(* CODESYS project Untitled2.project
   CustomField04_name: CustomField04
   CustomField06_name: CustomField06
   CustomField07_name: CustomField07
   CustomField09_name: CustomField09
   CustomField08_name: CustomField08
   CustomField02_name: CustomField02
   CustomField10_name: CustomField10
   CustomField01_name: CustomField01
   CustomField03_name: CustomField03
   CustomField05_name: CustomField05

Project tree, tasks and I/O mapping:
  MyController : TM258LF42DR, Schneider Electric, order no. TM258LF42DR, version 2.0.31.14
    application Application
      task MAST (cyclic, interval 20 ms, priority 15, watchdog 100 ms x 1) calls POU
      function HiddenPOU [ST]
      global variables GVL
      program POU [ST]
    Expert
      PowerDistribution : POWER, Schneider Electric, order no. POWER, version 2.0.31.14
          unmapped channels: IB0
      DM72F0 : DM72F0, Schneider Electric, order no. DM72F0, version 2.0.31.14
          settings: Synchronization.Output process task = 'MAST'
          unmapped channels: IB0, IB1, QB0
      DM72F1 : DM72F1, Schneider Electric, order no. DM72F1, version 2.0.31.14
          settings: Synchronization.Output process task = 'MAST'
          unmapped channels: IB0, IB1, QB0
    TM5
      TM5_Manager : TM5 Manager, Schneider Electric, order no. TM5, version 2.0.2.3
        Embedded Bus
          DI6DE : DI6DE, Schneider Electric, order no. DI6DE, version 3.1.1.1
              unmapped channels: DigitalInputs
          DI6DE_1 : DI6DE, Schneider Electric, order no. DI6DE, version 3.1.1.1
              unmapped channels: DigitalInputs
          DO6RE : DO6RE, Schneider Electric, order no. DO6RE, version 3.1.1.1
              unmapped channels: DigitalOutputs
          D000E : D000E, Schneider Electric, order no. D000E, version 3.1.1.1
          DO6RE_1 : DO6RE, Schneider Electric, order no. DO6RE, version 3.1.1.1
              unmapped channels: DigitalOutputs
    Ethernet
    Serial Line
      SoMachine_Network_Manager : SoMachine-Network_Manager, Schneider Electric, version 2.0.1.10
    CAN0
    PCI Slots
      <Empty>
      <Empty>
*)

// MyController/Application/GVL
VAR_GLOBAL
END_VAR

// MyController/Application/POU
PROGRAM POU
VAR
END_VAR

END_PROGRAM

// MyController/Application/HiddenPOU
FUNCTION HiddenPOU : BOOL

VAR_INPUT
	pHiddenFunc: POINTER TO WORD;
END_VAR
VAR
	pRead: POINTER TO BYTE;
	pWrite: POINTER TO BYTE;
END_VAR

pRead := pHiddenFunc + 400;
pWrite := pHiddenFunc + 4400;
HiddenPOU := TRUE;

END_FUNCTION
